SYSTEM ClientTest_2
  APPLICATION ClientTestApp
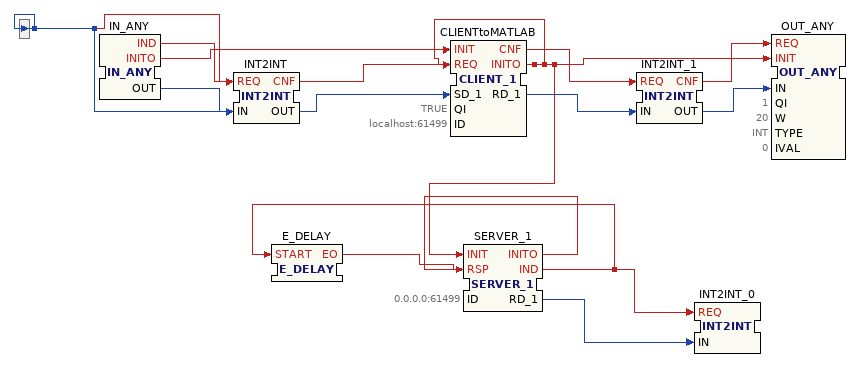
    FBS
      CLIENTtoMATLAB : CLIENT_1(QI := TRUE, ID := localhost:61499);
      INT2INT : INT2INT;
      OUT_ANY : OUT_ANY(QI := 1, W := 20, TYPE := INT, IVAL := 0);
      INT2INT_1 : INT2INT;
      IN_ANY : IN_ANY;
      SERVER_1 : SERVER_1(ID := 0.0.0.0:61499);
      INT2INT_0 : INT2INT;
      E_DELAY : E_DELAY;
    END_FBS
    EVENT_CONNECTIONS
       TO ;
       TO INT2INT.REQ;
      INT2INT_1.CNF TO OUT_ANY.REQ;
      IN_ANY.IND TO INT2INT.REQ;
      CLIENTtoMATLAB.CNF TO INT2INT_1.REQ;
      IN_ANY.INITO TO CLIENTtoMATLAB.INIT;
      CLIENTtoMATLAB.INITO TO OUT_ANY.INIT;
      INT2INT.CNF TO CLIENTtoMATLAB.REQ;
      CLIENTtoMATLAB.INITO TO CLIENTtoMATLAB.REQ;
      CLIENTtoMATLAB.INITO TO SERVER_1.INIT;
      SERVER_1.INITO TO SERVER_1.RSP;
      SERVER_1.IND TO INT2INT_0.REQ;
      SERVER_1.IND TO E_DELAY.START;
      E_DELAY.EO TO SERVER_1.RSP;
    END_CONNECTIONS
    DATA_CONNECTIONS
       TO INT2INT.IN;
       TO ;
      INT2INT_1.OUT TO OUT_ANY.IN;
      IN_ANY.OUT TO INT2INT.IN;
      CLIENTtoMATLAB.RD_1 TO INT2INT_1.IN;
      INT2INT.OUT TO CLIENTtoMATLAB.SD_1;
      SERVER_1.RD_1 TO INT2INT_0.IN;
    END_CONNECTIONS
  END_APPLICATION
  DEVICE CLIENT OBJECT : FORTE_PC(MGR_ID := "localhost:61499")
    {SET_ATTRIBUTE(Profile, HOLOBLOC)}
    RESOURCE EMB_RES_1 : EMB_RES
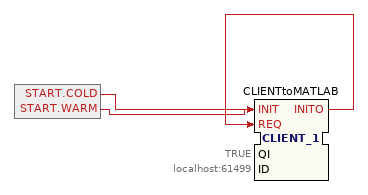
      FBS
        CLIENTtoMATLAB : CLIENT_1(QI := TRUE, ID := localhost:61499);
      END_FBS
      EVENT_CONNECTIONS
        START.COLD TO CLIENTtoMATLAB.INIT;
        START.WARM TO CLIENTtoMATLAB.INIT;
        CLIENTtoMATLAB.INITO TO CLIENTtoMATLAB.REQ;
      END_CONNECTIONS
    END_RESOURCE
  END_DEVICE
  DEVICE HMI : FBRT_WINDOW(MGR_ID := "localhost:61505")
    {SET_ATTRIBUTE(Profile, HOLOBLOC)}
    RESOURCE PANEL_RESOURCE : PANEL_RESOURCE
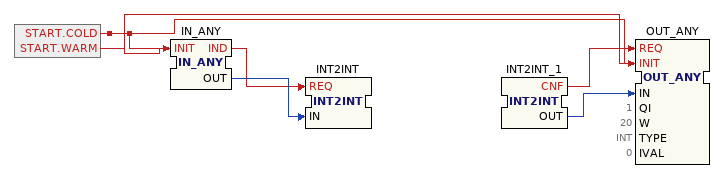
      FBS
        IN_ANY : IN_ANY;
        INT2INT : INT2INT;
        INT2INT_1 : INT2INT;
        OUT_ANY : OUT_ANY(QI := 1, W := 20, TYPE := INT, IVAL := 0);
      END_FBS
      EVENT_CONNECTIONS
        IN_ANY.IND TO INT2INT.REQ;
        INT2INT_1.CNF TO OUT_ANY.REQ;
        START.COLD TO IN_ANY.INIT;
        START.WARM TO IN_ANY.INIT;
        START.COLD TO OUT_ANY.INIT;
        START.WARM TO OUT_ANY.INIT;
      END_CONNECTIONS
      DATA_CONNECTIONS
        IN_ANY.OUT TO INT2INT.IN;
        INT2INT_1.OUT TO OUT_ANY.IN;
      END_CONNECTIONS
    END_RESOURCE
  END_DEVICE
  DEVICE FORTE_PC : FORTE_PC(MGR_ID := "0.0.0.0:61499")
    {SET_ATTRIBUTE(Profile, HOLOBLOC)}
    RESOURCE EMB_RES : EMB_RES
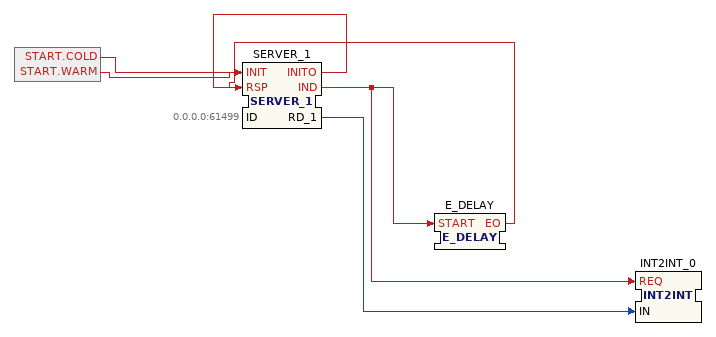
      FBS
        SERVER_1 : SERVER_1(ID := 0.0.0.0:61499);
        E_DELAY : E_DELAY;
        INT2INT_0 : INT2INT;
      END_FBS
      EVENT_CONNECTIONS
        START.COLD TO SERVER_1.INIT;
        START.WARM TO SERVER_1.INIT;
        SERVER_1.INITO TO SERVER_1.RSP;
        SERVER_1.IND TO E_DELAY.START;
        E_DELAY.EO TO SERVER_1.RSP;
        SERVER_1.IND TO INT2INT_0.REQ;
      END_CONNECTIONS
      DATA_CONNECTIONS
        SERVER_1.RD_1 TO INT2INT_0.IN;
      END_CONNECTIONS
    END_RESOURCE
  END_DEVICE
  MAPPINGS
    ClientTestApp.CLIENTtoMATLAB ON CLIENT OBJECT.EMB_RES_1.CLIENTtoMATLAB;
    ClientTestApp.INT2INT ON HMI.PANEL_RESOURCE.INT2INT;
    ClientTestApp.OUT_ANY ON HMI.PANEL_RESOURCE.OUT_ANY;
    ClientTestApp.INT2INT_1 ON HMI.PANEL_RESOURCE.INT2INT_1;
    ClientTestApp.IN_ANY ON HMI.PANEL_RESOURCE.IN_ANY;
    ClientTestApp.SERVER_1 ON FORTE_PC.EMB_RES.SERVER_1;
    ClientTestApp.INT2INT_0 ON FORTE_PC.EMB_RES.INT2INT_0;
    ClientTestApp.E_DELAY ON FORTE_PC.EMB_RES.E_DELAY;
  END_MAPPINGS
  SEGMENTS
    Ethernet : Ethernet;
  END_SEGMENTS
  LINKS
    CLIENT OBJECT => Ethernet;
    HMI => Ethernet;
    FORTE_PC => Ethernet;
  END_LINKS
END_SYSTEM
